Staubli VAL3: prgm1.pgx

program prgm1()
begin
  //while true
    //if(EntreePwrl0==true)
      open(tTool)
      movej(jP1, tTool, mNomSpeed)
      movej(jP2, tTool, mNomSpeed)
      close(tTool)
      movej(jP4, tTool, mNomSpeed)
      movej(jP5, tTool, mNomSpeed)
      movej(jP3, tTool, mNomSpeed)
      open(tTool)
      movej(jP1, tTool, mNomSpeed)
      movej(jP3, tTool, mNomSpeed)
      close(tTool)
      movej(jP5, tTool, mNomSpeed)
      movej(jP4, tTool, mNomSpeed)
      movej(jP2, tTool, mNomSpeed)
      open(tTool)
      waitEndMove()
    //endIf
 // endWhile
end
